# B&R Automation Studio project PLC_base3
Automation Studio 4.8.2.72

## Configuration Config1

CPU X20CP1382, AutomationRuntime B4.82, Build 4.1.2, Vc V4.72.1

### Task classes (Cpu.sw)
```
Cyclic#2:
  Program <- Program.prg
Binaries: udbdef, FWRules, TCData, sysconf, Role, User, iomap, ashwd, asfw, arconfig, ashwac
Libraries: standard, runtime, astime, asieccon
```

### Hardware
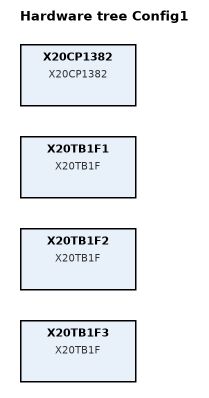
```
X20CP1382 : X20CP1382 v1.10.0.0  [X1 -> X1a.SL; X2 -> X2a.SL; X3 -> X3a.SL]
  Module X1a (Type=X1, Virtual=true, Version=1.10.0.0)
    Connection (Connector=SS1, TargetModule=X20TB1F1, TargetConnector=SS)
    Connection (Connector=SL, TargetModule=X20CP1382, TargetConnector=X1)
  Module X2a (Type=X2, Virtual=true, Version=1.10.0.0)
    Connection (Connector=SS1, TargetModule=X20TB1F2, TargetConnector=SS)
    Connection (Connector=SL, TargetModule=X20CP1382, TargetConnector=X2)
  Module X3a (Type=X3, Virtual=true, Version=1.10.0.0)
    Connection (Connector=SS1, TargetModule=X20TB1F3, TargetConnector=SS)
    Connection (Connector=SL, TargetModule=X20CP1382, TargetConnector=X3)
  Connector IF2:
    ActivateDevice = 1
    Mode = Manual
    InternetAddress = 192.168.0.69
    SubnetMask = 255.255.255.0
    ActivateSnmp = 2
  ConfigurationID = PLC_base3_Config1
  Simulation = 1
  SystemTick = 1000
  Cyclic1Duration = 1000
  Cyclic1Tolerance = 1000
X20TB1F1 : X20TB1F v1.0.0.0
X20TB1F2 : X20TB1F v1.0.0.0
X20TB1F3 : X20TB1F v1.0.0.0
```

### IoMap.iom - X20CP1382/IoMap.iom
```iecst
VAR_CONFIG
	::Program:enableX AT %QX."X3a".DigitalOutput01;
	::Program:enableY AT %QX."X3a".DigitalOutput02;
	::Program:enableZ AT %QX."X3a".DigitalOutput03;
	::Program:directionX AT %QX."X3a".DigitalOutput04;
	::Program:directionY AT %QX."X3a".DigitalOutput05;
	::Program:directionZ AT %QX."X3a".DigitalOutput06;
	::Program:bspidser AT %QX."X3a".DigitalOutput08;
	::Program:stepX AT %QX."X3a".DigitalOutput09;
	::Program:stepY AT %QX."X3a".DigitalOutput10;
	::Program:stepZ AT %QX."X3a".DigitalOutput11;
	::Program:stopZ AT %IX."X1a".DigitalInput01;
	::Program:stopY AT %IX."X1a".DigitalInput02;
	::Program:stopX AT %IX."X1a".DigitalInput03;
	::Program:stopB AT %IX."X1a".DigitalInput04;
END_VAR
```

## Logical view

Binary libraries used (declarations not repeated): operator, runtime, astime, AsIecCon, standard, AsBrStr, AsTCP


### Program Logical/Program (IEC)

#### Types.typ
```iecst
TYPE
	COMMSTATE2 :
		(
		RECEIVING,
		OFFLINE,
		EXECUTING,
		CONNECTED
		);
	ROBOSTATE2 :
		(
		CONVERT,
		STOP,
		MOVE0,
		NOT_DRAW,
		DRAW,
		BLYANTSPIDSER,
		MOVE_1,
		MOVE_2
		);
	STRING_ANALYZER :
		(
		STRING_ANALYZING,
		STRING_ANALYZE,
		STRING_ANALYZE_EM,
		STRING_ANALYZE_EMPTY_A
		);
	STRING_TOKENIZER :
		(
		STING_TOKEN
		);
	TCPSTATE2 :
		(
		TCPSTATE_SOCKET_CLOSE,
		TCPSTATE_SEND,
		TCPSTATE_SOCKET_OPEN,
		TCPSTATE_RECEIVE,
		TCPSTATE_SERVER_CREATE
		);
END_TYPE
```

#### Variables.var
```iecst
VAR
	COMMSTATE : COMMSTATE2;
	ROBOSTATE : ROBOSTATE2;
	count : UINT;
	bspidser : {REDUND_UNREPLICABLE} BOOL;
	enableX : {REDUND_UNREPLICABLE} BOOL;
	enableY : {REDUND_UNREPLICABLE} BOOL;
	enableZ : {REDUND_UNREPLICABLE} BOOL;
	directionX : BOOL;
	directionY : BOOL;
	directionZ : BOOL;
	stepX : BOOL;
	stepY : BOOL;
	stepZ : BOOL;
	stopB : BOOL;
	stopX : BOOL;
	stopY : BOOL;
	stopZ : BOOL;
	start1 : BOOL;
	timer : TON;
	A_KILL_SWITCH : BOOL;
END_VAR
(*STRING_TOKENIZER*)
VAR
	delim2 : STRING[80];
	delim1 : STRING[80];
	mainstring : STRING[80];
	x1 : INT;
	y1 : INT;
	x2 : INT;
	y2string : STRING[80];
	x2string : STRING[80];
	y1string : STRING[80];
	x1string : STRING[80];
	y2 : INT;
	string1 : STRING[80];
	string2 : STRING[80];
	D1 : INT;
	D2 : INT;
	D3 : INT;
	D4 : INT;
END_VAR
(*TCPSOCKET*)
VAR
	tcpstate : TCPSTATE2;
	tcpOpen1 : TcpOpen;
	tcpServer1 : TcpServer;
	tcpSend1 : TcpSend;
	tcpReceive1 : TcpRecv;
	tcpClose1 : TcpClose;
	tcpClose2 : TcpClose;
	receiveData : STRING[80];
	sendData : STRING[80];
END_VAR
(*STRING_ANALYZER*)
VAR
	stringState : STRING_ANALYZER;
	MoveX : INT;
	MoveY : INT;
	MoveZ : INT;
	value_countX : INT;
	value_countY : INT;
	value_countZ : INT;
END_VAR
(*MOVEMENT*)
VAR
	yPosPrev : INT;
	xPosPrev : INT;
	yPos : INT;
	xPos : INT;
	scale : INT;
END_VAR
```

#### LocalFunctions.fun
```iecst
{REDUND_ERROR} FUNCTION COORD_TO_STEP : INT (*Omdanner et koordinat til et antal steps*) (*$GROUP=User,$CAT=User,$GROUPICON=User.png,$CATICON=User.png*)
	VAR_INPUT
		COORD : UINT;
		SCALE : UINT;
	END_VAR
	VAR
		STEP_COUNT : UINT;
	END_VAR
END_FUNCTION
```

#### Main.st
```iecst
PROGRAM _INIT
	enableX := FALSE;
	enableY := FALSE;
	enableZ := FALSE;
	mainstring := '';

count:= 0;

END_PROGRAM

PROGRAM _CYCLIC
	IF A_KILL_SWITCH THEN			//Hvis noget går galt kan øverste variabel, denne, sættes TRUE/1 og motorerne slår fra.
	  ROBOSTATE := STOP;
	END_IF;

	(*CASE COMMSTATE OF
		CONNECTED:
		RECEIVING:

		OFFLINE:

	END_CASE;*)

	CASE tcpstate OF										//Socket communications
		TCPSTATE_SOCKET_OPEN:
			tcpOpen1.enable := TRUE;
			tcpOpen1.port := 80;
			tcpOpen1.options := tcpOPT_REUSEADDR;
			tcpOpen1();
			IF (tcpOpen1.status = ERR_OK) THEN
				tcpstate := TCPSTATE_SERVER_CREATE;
			END_IF;

		TCPSTATE_SERVER_CREATE:
			tcpServer1.enable := TRUE;
			tcpServer1.ident := tcpOpen1.ident;
			tcpServer1();
			IF (tcpServer1.status = ERR_OK) THEN
				tcpstate := TCPSTATE_RECEIVE;
			END_IF

		TCPSTATE_RECEIVE:
			tcpReceive1.enable := TRUE;
			tcpReceive1.ident := tcpServer1.identclnt;
			tcpReceive1.pData := ADR(receiveData);
			tcpReceive1.datamax := SIZEOF(receiveData);
			tcpReceive1();
			IF (tcpReceive1.status = ERR_OK) THEN
				tcpstate := TCPSTATE_SOCKET_CLOSE;
				sendData := '';
				sendData := LEFT(receiveData, UDINT_TO_INT(tcpReceive1.recvlen));
			END_IF

		(*TCPSTATE_SEND:
			tcpSend1.enable := TRUE;
			tcpSend1.ident := tcpServer1.identclnt;
			tcpSend1.pData := ADR(sendData);
			tcpSend1.datalen := brsstrlen (ADR(sendData));     // We use brsstrlen() to get the length in UDINT datatype
			tcpSend1();
			IF (tcpSend1.status = ERR_OK) THEN
				tcpstate := TCPSTATE_SOCKET_CLOSE;
			END_IF*)

		TCPSTATE_SOCKET_CLOSE:
			tcpClose1.enable := TRUE;
			tcpClose1.ident := tcpServer1.identclnt;
			tcpClose1();
			IF (tcpClose1.status = ERR_OK) THEN
				tcpServer1.enable := FALSE;
				tcpServer1();
				tcpstate := TCPSTATE_SERVER_CREATE;
			END_IF

	END_CASE;													//Socket communications end

	//StringTokenizer
	(*CASE Variable OF
		value:

	END_CASE;*)

	CASE ROBOSTATE OF								//Movement
		CONVERT:
			delim1 := ' ';
			delim2 := ',';

			//deler maintring i 2 strings med x og y i hver
			string1 := LEFT(mainstring, FIND(mainstring, delim2));
			string2 := RIGHT(mainstring, FIND(mainstring, delim2));

			//finder positioner af delimiters " " og "," i hver ny string
			D1 := FIND(string1, delim1);
			D2 := FIND(string1, delim2);
			D3 := FIND(string2, delim1);
			D4 := FIND(string2, delim2);

			x1string := LEFT(string1, D1 - 1);
			y1string := MID(string1, D2 - D1 - 1, D1 + 1);

			x2string := LEFT(string2, D3 - 1);
			y2string := MID(string2, D4 - D3 - 1, D3 + 1);

			//isolerer x og y koordinat i hver ny string
			x1 := STRING_TO_INT(x1string);
			y1 := STRING_TO_INT(y1string);

			x2 := STRING_TO_INT(x2string);
			y2 := STRING_TO_INT(y2string);

		STOP:
			enableX := TRUE;
			enableY := TRUE;
			enableZ := TRUE;

		MOVE_1:
			//bevæg sig efter x og y-koordinaterne
			xPos := x1;
			yPos := y1;

			MoveX := COORD_TO_STEP(xPos, scale) - COORD_TO_STEP(xPosPrev, scale);
			MoveY := COORD_TO_STEP(yPos, scale) - COORD_TO_STEP(yPosPrev, scale);
			xPosPrev := x1;
			yPosPrev := y1;
			xPos := x2;
			yPos := y2;

		MOVE_2:

			MoveX := COORD_TO_STEP(xPos, scale) - COORD_TO_STEP(xPosPrev, scale);
			MoveY := COORD_TO_STEP(yPos, scale) - COORD_TO_STEP(yPosPrev, scale);
			xPosPrev := x2;
			yPosPrev := y2;

		MOVE0:

			//bevæg sig til udgangsposition / origo

	(*	BLYANTSPIDSER:
			IF   start1 = TRUE THEN

		IF stopZ = FALSE AND stopX = FALSE THEN
			directionZ := FALSE;
	  		stepZ := NOT stepZ;
		END_IF;

		IF stopX = FALSE AND stopZ = TRUE THEN
			IF stepX = FALSE THEN
				stepX := TRUE;
			ELSIF
				stepX = TRUE THEN
				stepX := FALSE;

			END_IF;
	    	stepX := NOT stepX;
		END_IF;

		IF stopB = FALSE AND stopX = TRUE THEN
			directionZ := TRUE;
			stepZ := NOT stepZ;
		END_IF;

		timer.IN := NOT timer.Q;
		timer.PT := T#5s;
		timer();
		bspidser := timer.Q;

		IF stopZ = FALSE THEN
			directionZ := FALSE;
			stepZ := NOT stepZ;
		END_IF;

	END_IF;
		*)

		DRAW:
			WHILE NOT stopB DO
				directionZ := TRUE;
				stepZ := NOT stepZ;
			END_WHILE;

		NOT_DRAW:
			WHILE NOT stopZ DO
				directionZ := FALSE;
	  			stepZ := NOT stepZ;
			END_WHILE;

	END_CASE;

(*	IF start1 = TRUE THEN			//test til at køre fra ene side til anden på x-aksen og beregne længden fra pixel til praksis

		IF stopX = FALSE THEN
			stepX := NOT stepX;
			count := count + 1;
		END_IF

		IF stopX = TRUE THEN
	  		start1 := FALSE;
		END_IF;

	END_IF;		*)					//slut

END_PROGRAM

PROGRAM _EXIT
	tcpClose1.enable := TRUE;
	tcpClose1.ident := tcpServer1.identclnt;
	tcpClose1();

	tcpClose2.enable := TRUE;
	tcpClose2.ident := tcpOpen1.ident;
	tcpClose2();

END_PROGRAM
```

Listed in the project but not available here: Logical/Global.typ, Logical/Global.var
